// TIA Portal V20 export
FUNCTION_BLOCK "CallAlarmCounter"   // FB5, LAD
// stored: MemoryReserve 100, SetENOAutomatically false
   VAR
      statPulse { ExternalAccessible := 'False'; ExternalVisible := 'False'; ExternalWritable := 'False'} : Array[0..99] of Bool;
   END_VAR
   VAR_TEMP
      tempEnter : Bool;   // Enter the conditions for the count to increase.
   END_VAR
   VAR_TEMP   // added for the SCL form of the ladder/FBD networks
      _w1 : Bool;
   END_VAR
BEGIN

REGION Network 1: Counter Setting Save
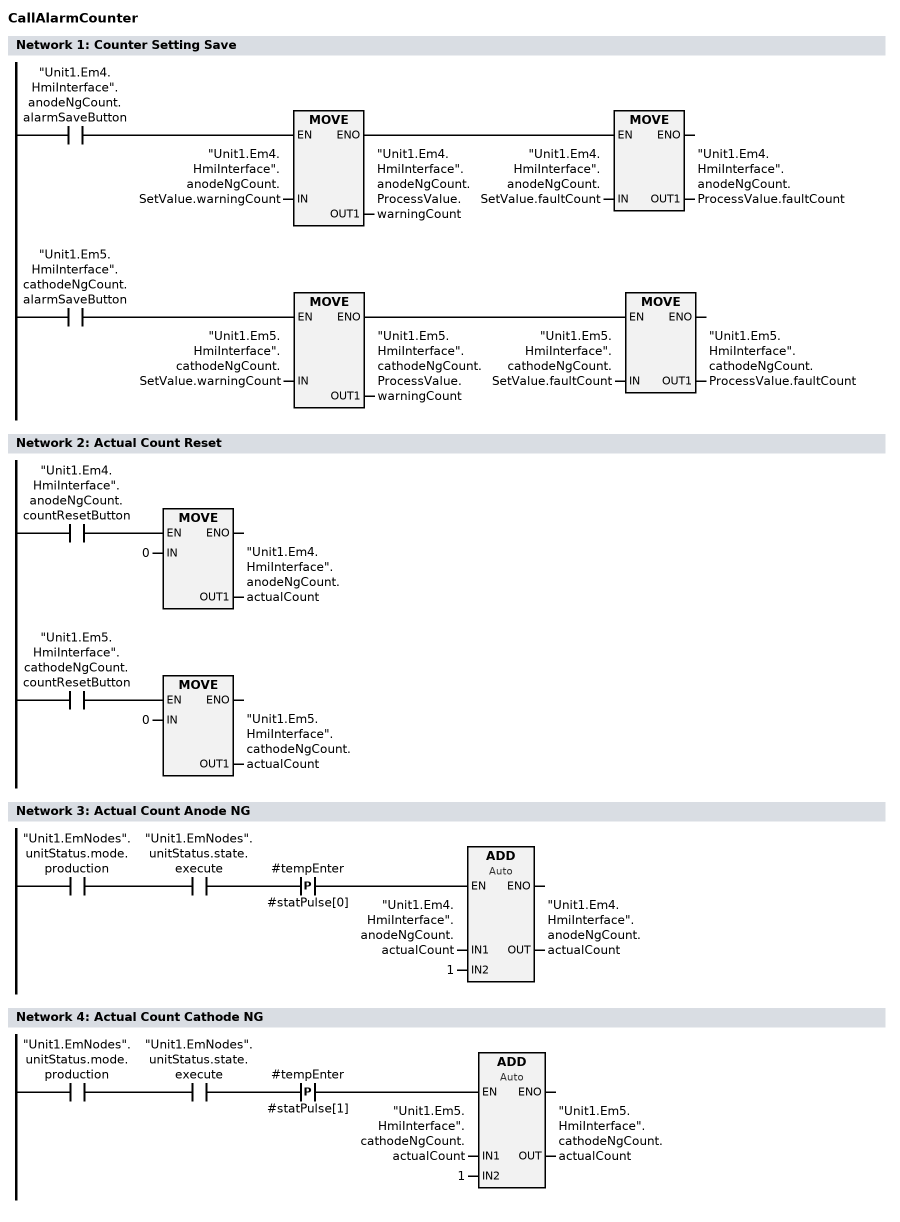
   RUNG wire#powerrail
      Contact( "Unit1.Em4.HmiInterface".anodeNgCount.alarmSaveButton )
      Move(in := "Unit1.Em4.HmiInterface".anodeNgCount.SetValue.warningCount, out1 => "Unit1.Em4.HmiInterface".anodeNgCount.ProcessValue.warningCount)
      Move(in := "Unit1.Em4.HmiInterface".anodeNgCount.SetValue.faultCount, out1 => "Unit1.Em4.HmiInterface".anodeNgCount.ProcessValue.faultCount)
   END_RUNG
   RUNG wire#powerrail
      Contact( "Unit1.Em5.HmiInterface".cathodeNgCount.alarmSaveButton )
      Move(in := "Unit1.Em5.HmiInterface".cathodeNgCount.SetValue.warningCount, out1 => "Unit1.Em5.HmiInterface".cathodeNgCount.ProcessValue.warningCount)
      Move(in := "Unit1.Em5.HmiInterface".cathodeNgCount.SetValue.faultCount, out1 => "Unit1.Em5.HmiInterface".cathodeNgCount.ProcessValue.faultCount)
   END_RUNG
   // the same network as SCL:
   IF "Unit1.Em4.HmiInterface".anodeNgCount.alarmSaveButton THEN
       "Unit1.Em4.HmiInterface".anodeNgCount.ProcessValue.warningCount := "Unit1.Em4.HmiInterface".anodeNgCount.SetValue.warningCount;
       "Unit1.Em4.HmiInterface".anodeNgCount.ProcessValue.faultCount := "Unit1.Em4.HmiInterface".anodeNgCount.SetValue.faultCount;
   END_IF;
   IF "Unit1.Em5.HmiInterface".cathodeNgCount.alarmSaveButton THEN
       "Unit1.Em5.HmiInterface".cathodeNgCount.ProcessValue.warningCount := "Unit1.Em5.HmiInterface".cathodeNgCount.SetValue.warningCount;
       "Unit1.Em5.HmiInterface".cathodeNgCount.ProcessValue.faultCount := "Unit1.Em5.HmiInterface".cathodeNgCount.SetValue.faultCount;
   END_IF;
END_REGION

REGION Network 2: Actual Count Reset
   RUNG wire#powerrail
      Contact( "Unit1.Em4.HmiInterface".anodeNgCount.countResetButton )
      Move(in := 0, out1 => "Unit1.Em4.HmiInterface".anodeNgCount.actualCount)
   END_RUNG
   RUNG wire#powerrail
      Contact( "Unit1.Em5.HmiInterface".cathodeNgCount.countResetButton )
      Move(in := 0, out1 => "Unit1.Em5.HmiInterface".cathodeNgCount.actualCount)
   END_RUNG
   // the same network as SCL:
   IF "Unit1.Em4.HmiInterface".anodeNgCount.countResetButton THEN
       "Unit1.Em4.HmiInterface".anodeNgCount.actualCount := 0;
   END_IF;
   IF "Unit1.Em5.HmiInterface".cathodeNgCount.countResetButton THEN
       "Unit1.Em5.HmiInterface".cathodeNgCount.actualCount := 0;
   END_IF;
END_REGION

REGION Network 3: Actual Count Anode NG
   RUNG wire#powerrail
      Contact( "Unit1.EmNodes".unitStatus.mode.production )
      Contact( "Unit1.EmNodes".unitStatus.state.execute )
      P_Contact(operand := #tempEnter, bit := #statPulse[0])
      Add(in1 := "Unit1.Em4.HmiInterface".anodeNgCount.actualCount, in2 := 1, out => "Unit1.Em4.HmiInterface".anodeNgCount.actualCount)
   END_RUNG
   // the same network as SCL:
   #_w1 := "Unit1.EmNodes".unitStatus.mode.production AND "Unit1.EmNodes".unitStatus.state.execute AND #tempEnter AND NOT #statPulse[0];   // rising edge of #tempEnter
   #statPulse[0] := #tempEnter;
   IF #_w1 THEN
       "Unit1.Em4.HmiInterface".anodeNgCount.actualCount := "Unit1.Em4.HmiInterface".anodeNgCount.actualCount + 1;
   END_IF;
END_REGION

REGION Network 4: Actual Count Cathode NG
   RUNG wire#powerrail
      Contact( "Unit1.EmNodes".unitStatus.mode.production )
      Contact( "Unit1.EmNodes".unitStatus.state.execute )
      P_Contact(operand := #tempEnter, bit := #statPulse[1])
      Add(in1 := "Unit1.Em5.HmiInterface".cathodeNgCount.actualCount, in2 := 1, out => "Unit1.Em5.HmiInterface".cathodeNgCount.actualCount)
   END_RUNG
   // the same network as SCL:
   #_w1 := "Unit1.EmNodes".unitStatus.mode.production AND "Unit1.EmNodes".unitStatus.state.execute AND #tempEnter AND NOT #statPulse[1];   // rising edge of #tempEnter
   #statPulse[1] := #tempEnter;
   IF #_w1 THEN
       "Unit1.Em5.HmiInterface".cathodeNgCount.actualCount := "Unit1.Em5.HmiInterface".cathodeNgCount.actualCount + 1;
   END_IF;
END_REGION
END_FUNCTION_BLOCK
